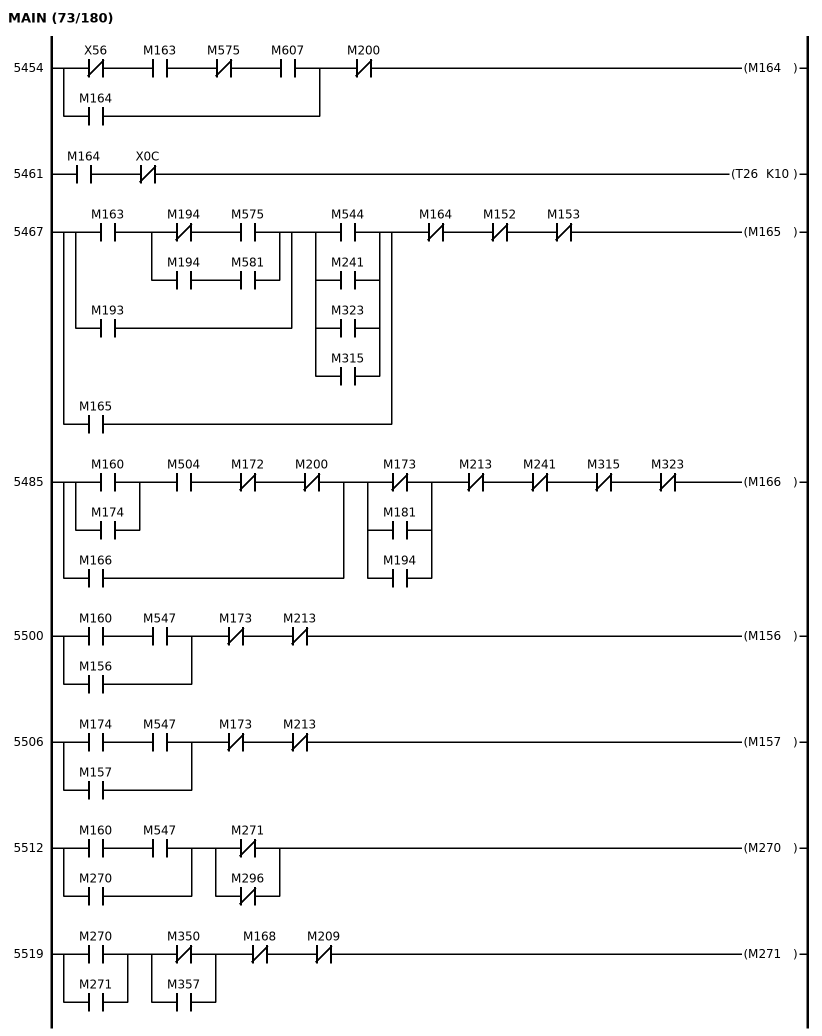
[picture p72: ladder of MAIN, rungs at steps 5454 to 5519]
5454  LDI     X56
      AND     M163
      ANI     M575
      AND     M607
      OR      M164
      ANI     M200
      OUT     M164
5461  LD      M164
      ANI     X0C
      OUT     T26 K10
5467  LD      M163
      LDI     M194
      AND     M575
      LD      M194
      AND     M581
      ORB
      ANB
      OR      M193
      LD      M544
      OR      M241
      OR      M323
      OR      M315
      ANB
      OR      M165
      ANI     M164
      ANI     M152
      ANI     M153
      OUT     M165
5485  LD      M160
      OR      M174
      AND     M504
      ANI     M172
      ANI     M200
      OR      M166
      LDI     M173
      OR      M181
      OR      M194
      ANB
      ANI     M213
      ANI     M241
      ANI     M315
      ANI     M323
      OUT     M166
5500  LD      M160
      AND     M547
      OR      M156
      ANI     M173
      ANI     M213
      OUT     M156
5506  LD      M174
      AND     M547
      OR      M157
      ANI     M173
      ANI     M213
      OUT     M157
5512  LD      M160
      AND     M547
      OR      M270
      LDI     M271
      ORI     M296
      ANB
      OUT     M270
5519  LD      M270
      OR      M271
      LDI     M350
      OR      M357
      ANB
      ANI     M168
      ANI     M209
      OUT     M271
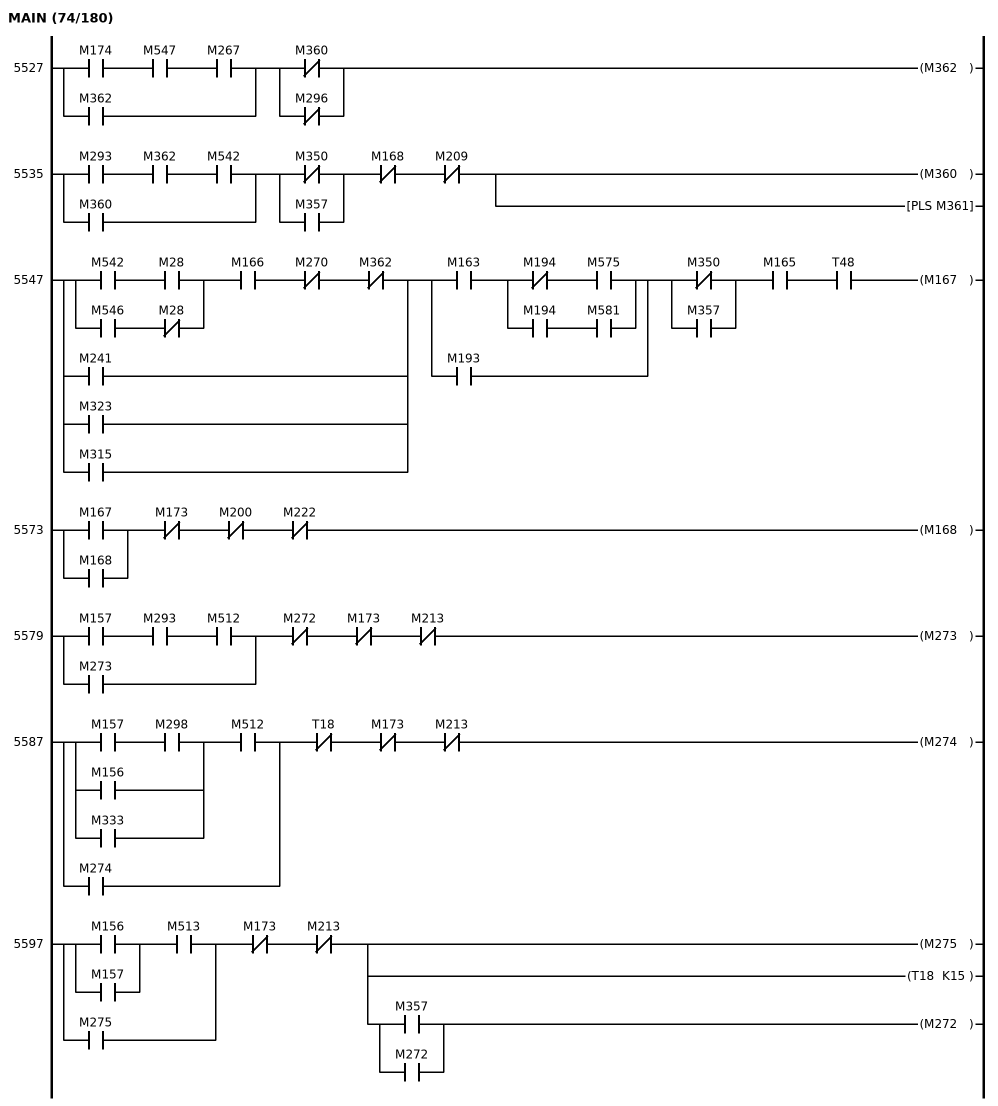
5527  LD      M174
      AND     M547
      AND     M267
      OR      M362
      LDI     M360
      ORI     M296
      ANB
      OUT     M362
5535  LD      M293
      AND     M362
      AND     M542
      OR      M360
      LDI     M350
      OR      M357
      ANB
      ANI     M168
      ANI     M209
      OUT     M360
      PLS     M361
5547  LD      M542
      AND     M28
      LD      M546
      ANI     M28
      ORB
      AND     M166
      ANI     M270
      ANI     M362
      OR      M241
      OR      M323
      OR      M315
      LD      M163
      LDI     M194
      AND     M575
      LD      M194
      AND     M581
      ORB
      ANB
      OR      M193
      ANB
      LDI     M350
      OR      M357
      ANB
      AND     M165
      AND     T48
      OUT     M167
5573  LD      M167
      OR      M168
      ANI     M173
      ANI     M200
      ANI     M222
      OUT     M168
5579  LD      M157
      AND     M293
      AND     M512
      OR      M273
      ANI     M272
      ANI     M173
      ANI     M213
      OUT     M273
5587  LD      M157
      AND     M298
      OR      M156
      OR      M333
      AND     M512
      OR      M274
      ANI     T18
      ANI     M173
      ANI     M213
      OUT     M274
5597  LD      M156
      OR      M157
      AND     M513
      OR      M275
      ANI     M173
      ANI     M213
      OUT     M275
      OUT     T18 K15
      LD      M357
      OR      M272
      ANB
      OUT     M272
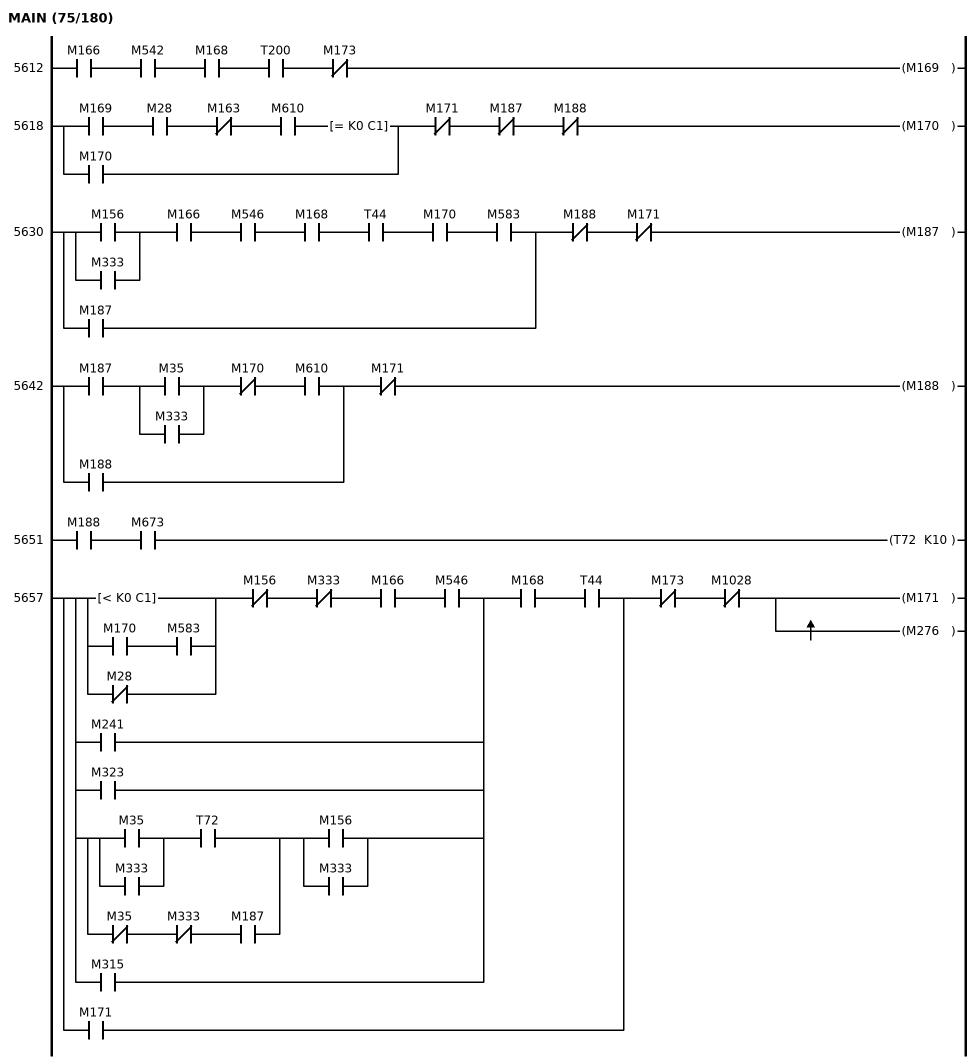
5612  LD      M166
      AND     M542
      AND     M168
      AND     T200
      ANI     M173
      OUT     M169
5618  LD      M169
      AND     M28
      ANI     M163
      AND     M610
      AND=    K0 C1
      OR      M170
      ANI     M171
      ANI     M187
      ANI     M188
      OUT     M170
5630  LD      M156
      OR      M333
      AND     M166
      AND     M546
      AND     M168
      AND     T44
      AND     M170
      AND     M583
      OR      M187
      ANI     M188
      ANI     M171
      OUT     M187
5642  LD      M187
      LD      M35
      OR      M333
      ANB
      ANI     M170
      AND     M610
      OR      M188
      ANI     M171
      OUT     M188
5651  LD      M188
      AND     M673
      OUT     T72 K10
5657  LD<     K0 C1
      LD      M170
      AND     M583
      ORB
      ORI     M28
      ANI     M156
      ANI     M333
      AND     M166
      AND     M546
      OR      M241
      OR      M323
      LD      M35
      OR      M333
      AND     T72
      LDI     M35
      ANI     M333
      AND     M187
      ORB
      LD      M156
      OR      M333
      ANB
      ORB
      OR      M315
      AND     M168
      AND     T44
      OR      M171
      ANI     M173
      ANI     M1028
      OUT     M171
      MEP
      OUT     M276
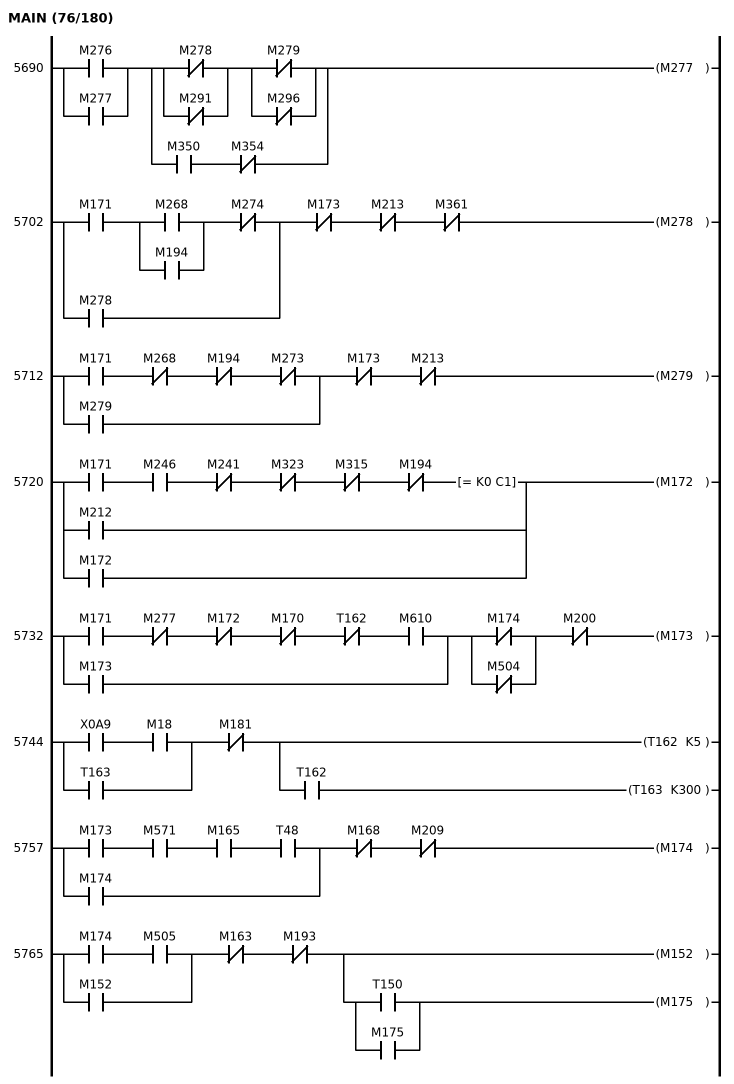
5690  LD      M276
      OR      M277
      LDI     M278
      ORI     M291
      LDI     M279
      ORI     M296
      ANB
      LD      M350
      ANI     M354
      ORB
      ANB
      OUT     M277
5702  LD      M171
      LD      M268
      OR      M194
      ANB
      ANI     M274
      OR      M278
      ANI     M173
      ANI     M213
      ANI     M361
      OUT     M278
5712  LD      M171
      ANI     M268
      ANI     M194
      ANI     M273
      OR      M279
      ANI     M173
      ANI     M213
      OUT     M279
5720  LD      M171
      AND     M246
      ANI     M241
      ANI     M323
      ANI     M315
      ANI     M194
      AND=    K0 C1
      OR      M212
      OR      M172
      OUT     M172
5732  LD      M171
      ANI     M277
      ANI     M172
      ANI     M170
      ANI     T162
      AND     M610
      OR      M173
      LDI     M174
      ORI     M504
      ANB
      ANI     M200
      OUT     M173
5744  LD      X0A9
      AND     M18
      OR      T163
      ANI     M181
      OUT     T162 K5
      AND     T162
      OUT     T163 K300
5757  LD      M173
      AND     M571
      AND     M165
      AND     T48
      OR      M174
      ANI     M168
      ANI     M209
      OUT     M174
5765  LD      M174
      AND     M505
      OR      M152
      ANI     M163
      ANI     M193
      OUT     M152
      LD      T150
      OR      M175
      ANB
      OUT     M175
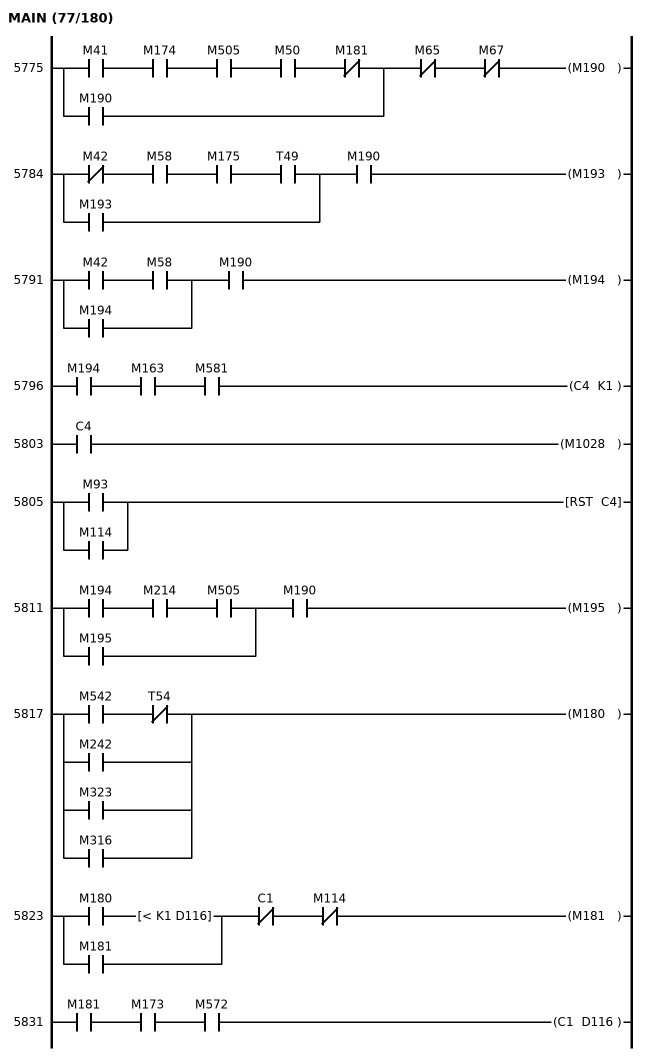
5775  LD      M41
      AND     M174
      AND     M505
      AND     M50
      ANI     M181
      OR      M190
      ANI     M65
      ANI     M67
      OUT     M190
5784  LDI     M42
      AND     M58
      AND     M175
      AND     T49
      OR      M193
      AND     M190
      OUT     M193
5791  LD      M42
      AND     M58
      OR      M194
      AND     M190
      OUT     M194
5796  LD      M194
      AND     M163
      AND     M581
      OUT     C4 K1
5803  LD      C4
      OUT     M1028
5805  LD      M93
      OR      M114
      RST     C4
5811  LD      M194
      AND     M214
      AND     M505
      OR      M195
      AND     M190
      OUT     M195
5817  LD      M542
      ANI     T54
      OR      M242
      OR      M323
      OR      M316
      OUT     M180
5823  LD      M180
      AND<    K1 D116
      OR      M181
      ANI     C1
      ANI     M114
      OUT     M181
5831  LD      M181
      AND     M173
      AND     M572
      OUT     C1 D116
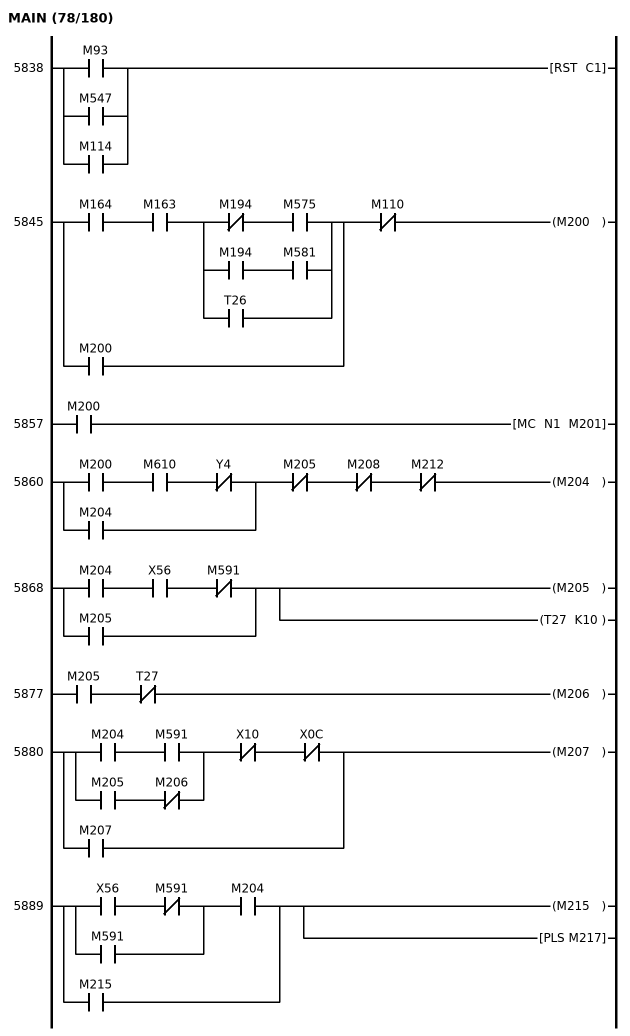
5838  LD      M93
      OR      M547
      OR      M114
      RST     C1
5845  LD      M164
      AND     M163
      LDI     M194
      AND     M575
      LD      M194
      AND     M581
      ORB
      OR      T26
      ANB
      OR      M200
      ANI     M110
      OUT     M200
5857  LD      M200
      MC      N1 M201
5860  LD      M200
      AND     M610
      ANI     Y4
      OR      M204
      ANI     M205
      ANI     M208
      ANI     M212
      OUT     M204
5868  LD      M204
      AND     X56
      ANI     M591
      OR      M205
      OUT     M205
      OUT     T27 K10
5877  LD      M205
      ANI     T27
      OUT     M206
5880  LD      M204
      AND     M591
      LD      M205
      ANI     M206
      ORB
      ANI     X10
      ANI     X0C
      OR      M207
      OUT     M207
5889  LD      X56
      ANI     M591
      OR      M591
      AND     M204
      OR      M215
      OUT     M215
      PLS     M217
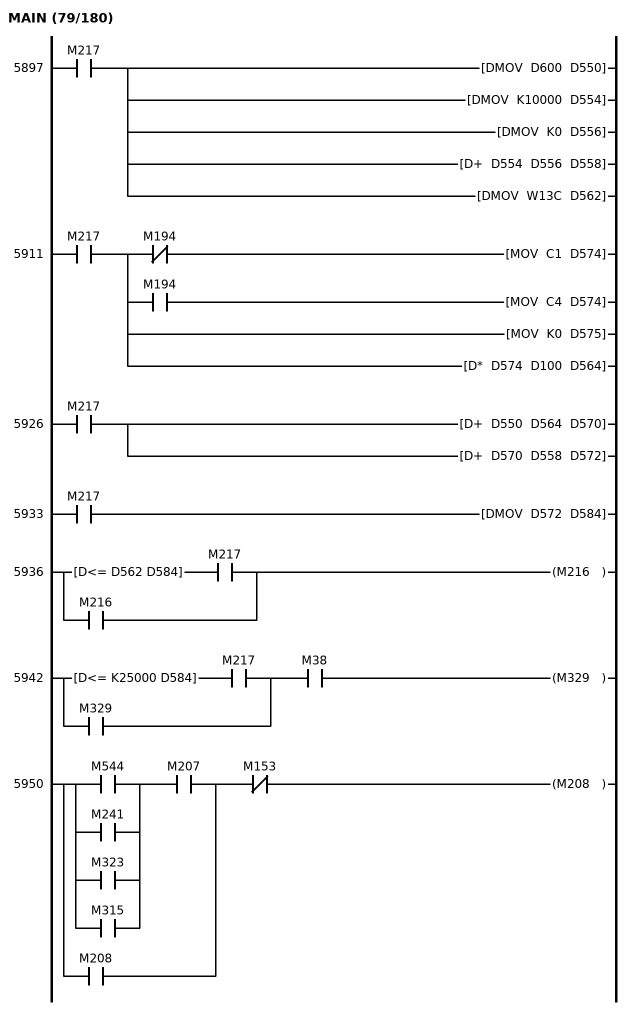
5897  LD      M217
      DMOV    D600 D550
      DMOV    K10000 D554
      DMOV    K0 D556
      D+      D554 D556 D558
      DMOV    W13C D562
5911  LD      M217
      MPS
      ANI     M194
      MOV     C1 D574
      MRD
      AND     M194
      MOV     C4 D574
      MPP
      MOV     K0 D575
      D*      D574 D100 D564
5926  LD      M217
      D+      D550 D564 D570
      D+      D570 D558 D572
5933  LD      M217
      DMOV    D572 D584
5936  LDD<=   D562 D584
      AND     M217
      OR      M216
      OUT     M216
5942  LDD<=   K25000 D584
      AND     M217
      OR      M329
      AND     M38
      OUT     M329
5950  LD      M544
      OR      M241
      OR      M323
      OR      M315
      AND     M207
      OR      M208
      ANI     M153
      OUT     M208
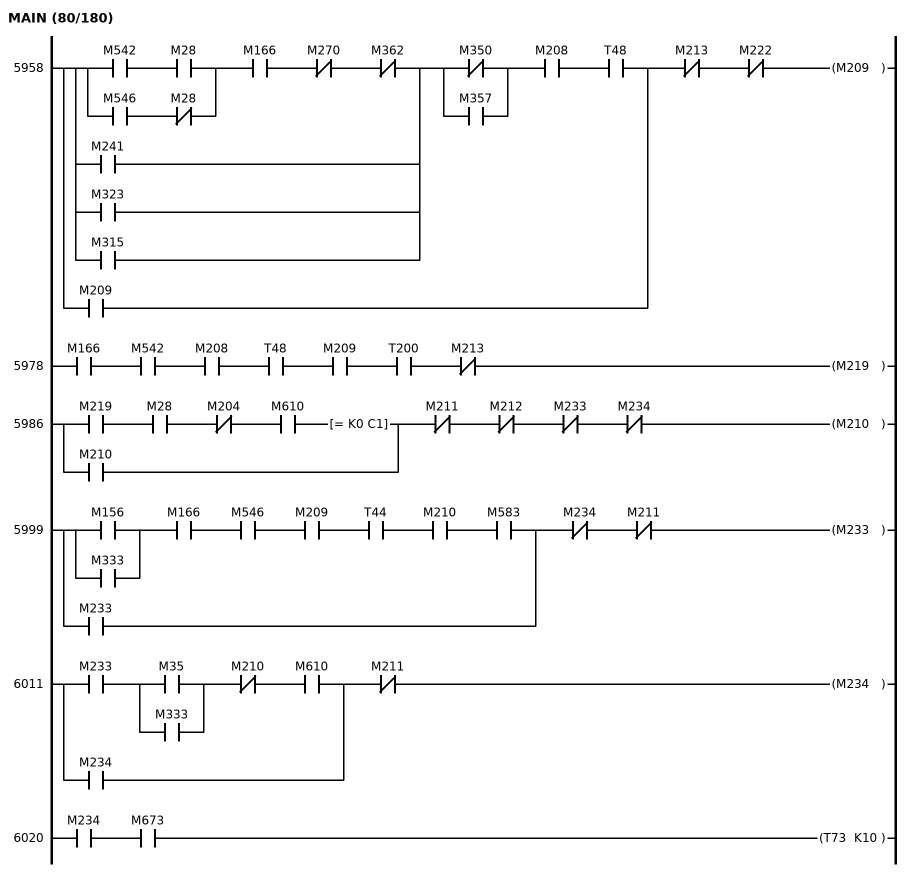
5958  LD      M542
      AND     M28
      LD      M546
      ANI     M28
      ORB
      AND     M166
      ANI     M270
      ANI     M362
      OR      M241
      OR      M323
      OR      M315
      LDI     M350
      OR      M357
      ANB
      AND     M208
      AND     T48
      OR      M209
      ANI     M213
      ANI     M222
      OUT     M209
5978  LD      M166
      AND     M542
      AND     M208
      AND     T48
      AND     M209
      AND     T200
      ANI     M213
      OUT     M219
5986  LD      M219
      AND     M28
      ANI     M204
      AND     M610
      AND=    K0 C1
      OR      M210
      ANI     M211
      ANI     M212
      ANI     M233
      ANI     M234
      OUT     M210
5999  LD      M156
      OR      M333
      AND     M166
      AND     M546
      AND     M209
      AND     T44
      AND     M210
      AND     M583
      OR      M233
      ANI     M234
      ANI     M211
      OUT     M233
6011  LD      M233
      LD      M35
      OR      M333
      ANB
      ANI     M210
      AND     M610
      OR      M234
      ANI     M211
      OUT     M234
6020  LD      M234
      AND     M673
      OUT     T73 K10
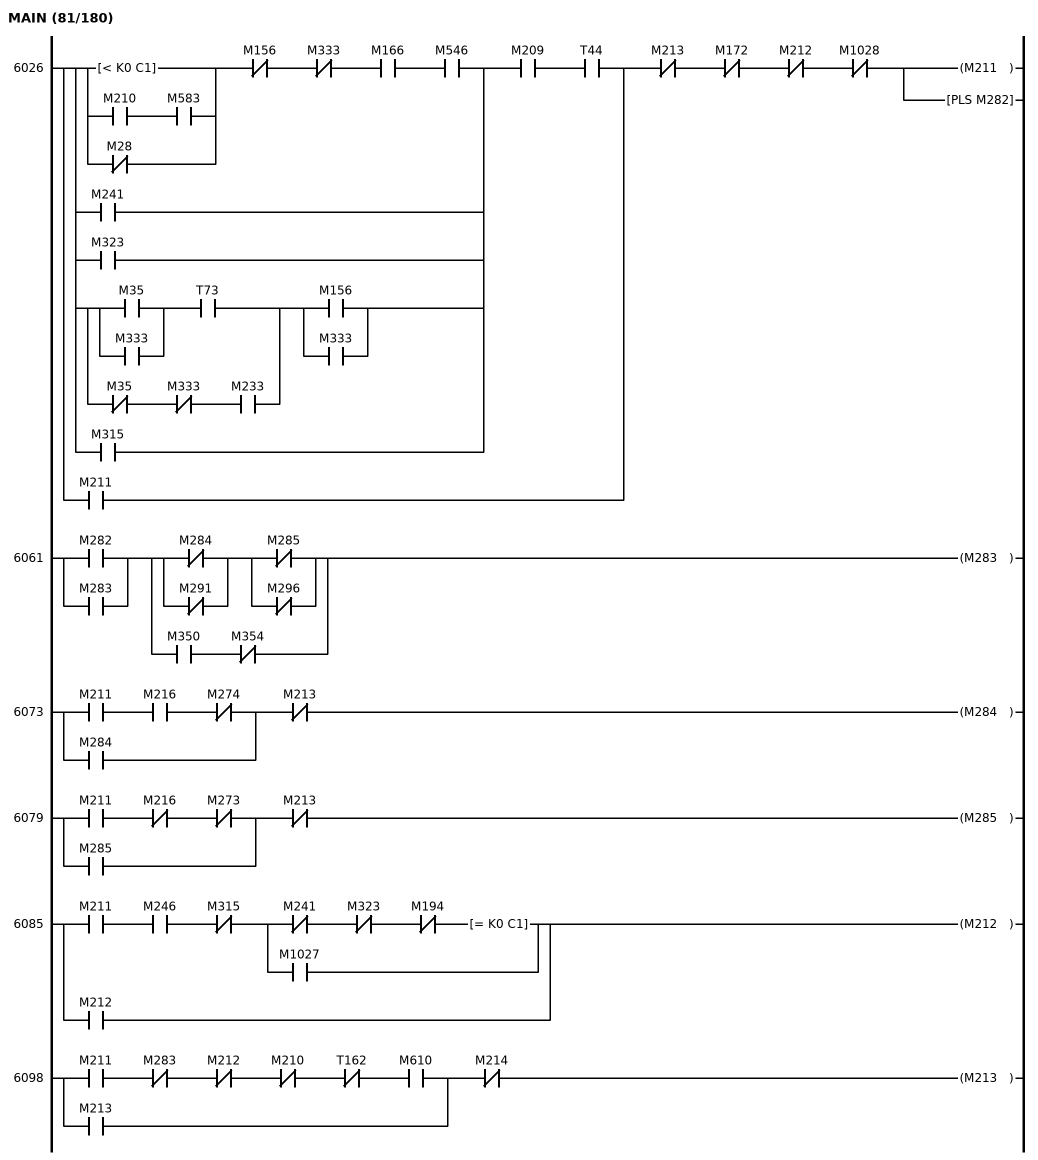
6026  LD<     K0 C1
      LD      M210
      AND     M583
      ORB
      ORI     M28
      ANI     M156
      ANI     M333
      AND     M166
      AND     M546
      OR      M241
      OR      M323
      LD      M35
      OR      M333
      AND     T73
      LDI     M35
      ANI     M333
      AND     M233
      ORB
      LD      M156
      OR      M333
      ANB
      ORB
      OR      M315
      AND     M209
      AND     T44
      OR      M211
      ANI     M213
      ANI     M172
      ANI     M212
      ANI     M1028
      OUT     M211
      PLS     M282
6061  LD      M282
      OR      M283
      LDI     M284
      ORI     M291
      LDI     M285
      ORI     M296
      ANB
      LD      M350
      ANI     M354
      ORB
      ANB
      OUT     M283
6073  LD      M211
      AND     M216
      ANI     M274
      OR      M284
      ANI     M213
      OUT     M284
6079  LD      M211
      ANI     M216
      ANI     M273
      OR      M285
      ANI     M213
      OUT     M285
6085  LD      M211
      AND     M246
      ANI     M315
      LDI     M241
      ANI     M323
      ANI     M194
      AND=    K0 C1
      OR      M1027
      ANB
      OR      M212
      OUT     M212
6098  LD      M211
      ANI     M283
      ANI     M212
      ANI     M210
      ANI     T162
      AND     M610
      OR      M213
      ANI     M214
      OUT     M213
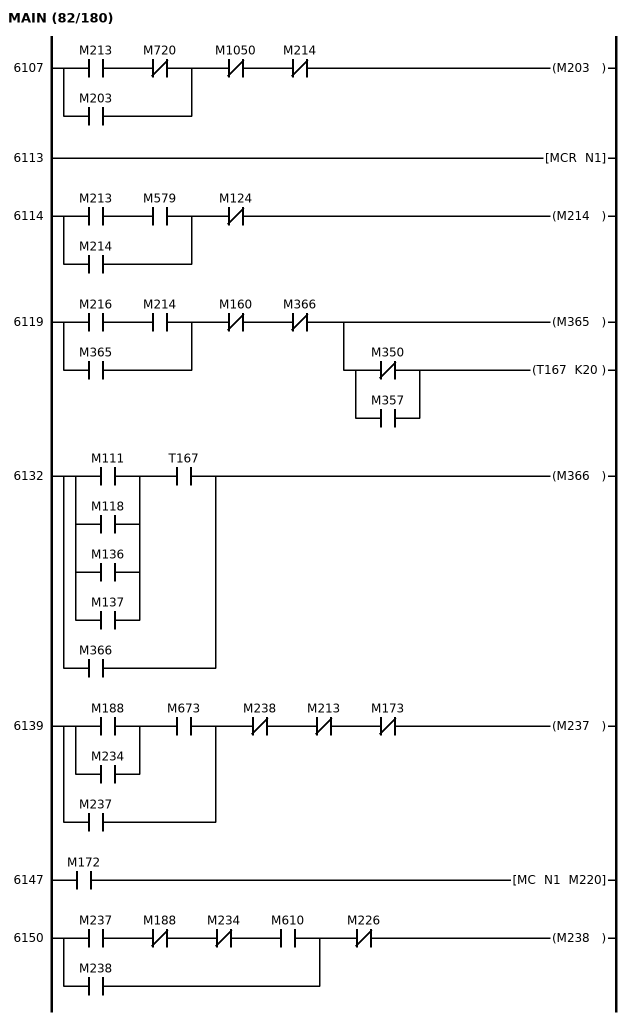
6107  LD      M213
      ANI     M720
      OR      M203
      ANI     M1050
      ANI     M214
      OUT     M203
6113  MCR     N1
6114  LD      M213
      AND     M579
      OR      M214
      ANI     M124
      OUT     M214
6119  LD      M216
      AND     M214
      OR      M365
      ANI     M160
      ANI     M366
      OUT     M365
      LDI     M350
      OR      M357
      ANB
      OUT     T167 K20
6132  LD      M111
      OR      M118
      OR      M136
      OR      M137
      AND     T167
      OR      M366
      OUT     M366
6139  LD      M188
      OR      M234
      AND     M673
      OR      M237
      ANI     M238
      ANI     M213
      ANI     M173
      OUT     M237
6147  LD      M172
      MC      N1 M220
6150  LD      M237
      ANI     M188
      ANI     M234
      AND     M610
      OR      M238
      ANI     M226
      OUT     M238
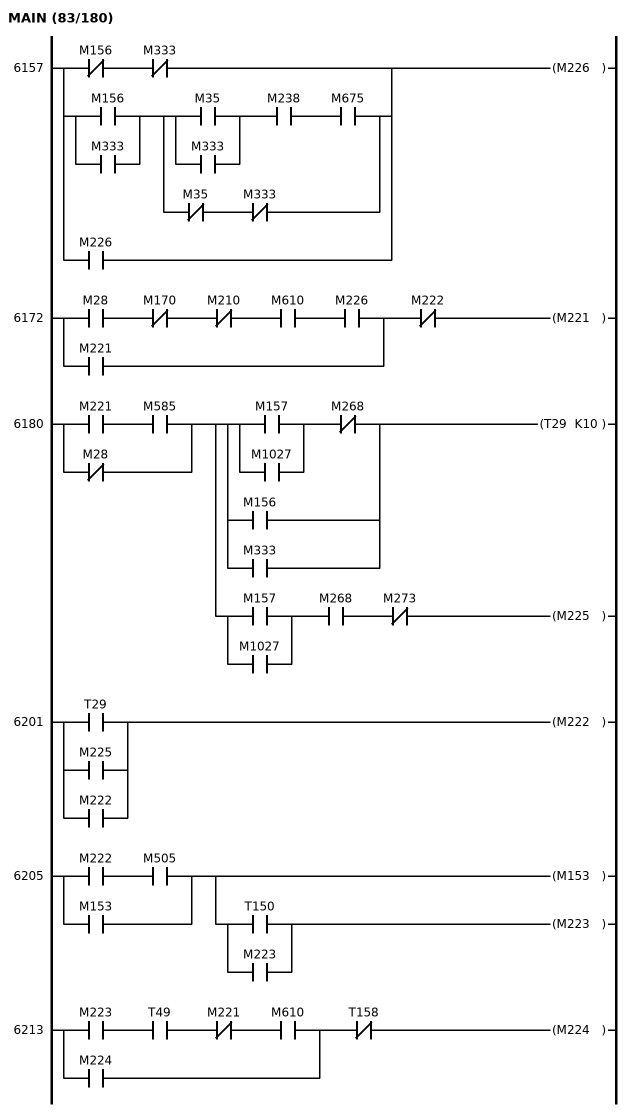
6157  LDI     M156
      ANI     M333
      LD      M156
      OR      M333
      LD      M35
      OR      M333
      AND     M238
      AND     M675
      LDI     M35
      ANI     M333
      ORB
      ANB
      ORB
      OR      M226
      OUT     M226
6172  LD      M28
      ANI     M170
      ANI     M210
      AND     M610
      AND     M226
      OR      M221
      ANI     M222
      OUT     M221
6180  LD      M221
      AND     M585
      ORI     M28
      MPS
      LD      M157
      OR      M1027
      ANI     M268
      OR      M156
      OR      M333
      ANB
      OUT     T29 K10
      MPP
      LD      M157
      OR      M1027
      ANB
      AND     M268
      ANI     M273
      OUT     M225
6201  LD      T29
      OR      M225
      OR      M222
      OUT     M222
6205  LD      M222
      AND     M505
      OR      M153
      OUT     M153
      LD      T150
      OR      M223
      ANB
      OUT     M223
6213  LD      M223
      AND     T49
      ANI     M221
      AND     M610
      OR      M224
      ANI     T158
      OUT     M224
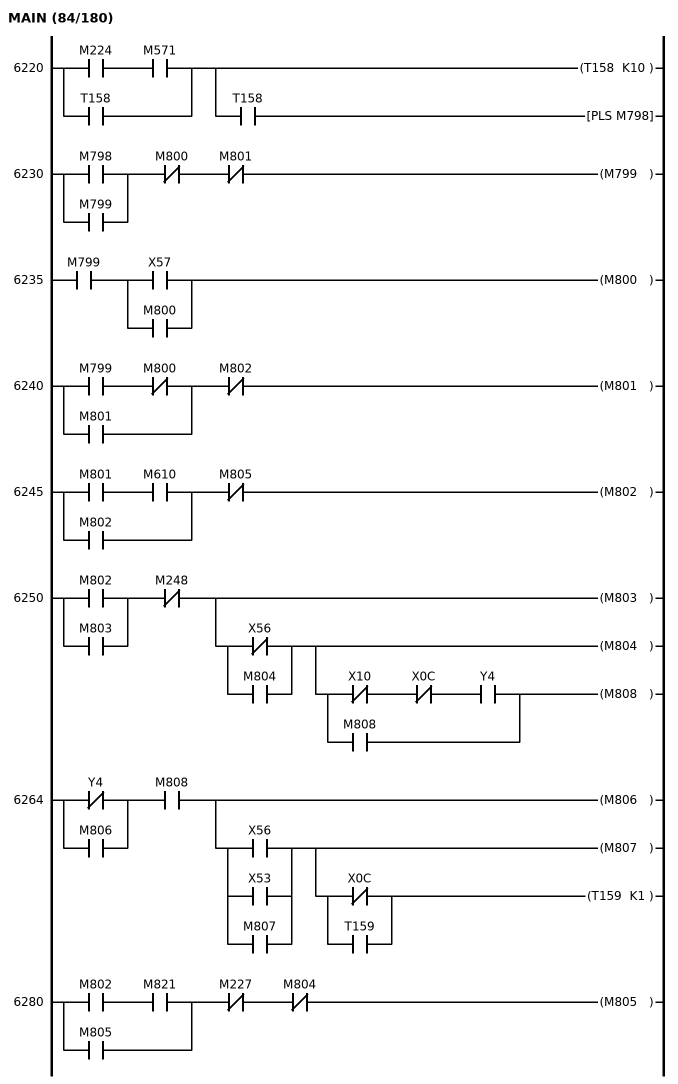
6220  LD      M224
      AND     M571
      OR      T158
      OUT     T158 K10
      AND     T158
      PLS     M798
6230  LD      M798
      OR      M799
      ANI     M800
      ANI     M801
      OUT     M799
6235  LD      M799
      LD      X57
      OR      M800
      ANB
      OUT     M800
6240  LD      M799
      ANI     M800
      OR      M801
      ANI     M802
      OUT     M801
6245  LD      M801
      AND     M610
      OR      M802
      ANI     M805
      OUT     M802
6250  LD      M802
      OR      M803
      ANI     M248
      OUT     M803
      LDI     X56
      OR      M804
      ANB
      OUT     M804
      LDI     X10
      ANI     X0C
      AND     Y4
      OR      M808
      ANB
      OUT     M808
6264  LDI     Y4
      OR      M806
      AND     M808
      OUT     M806
      LD      X56
      OR      X53
      OR      M807
      ANB
      OUT     M807
      LDI     X0C
      OR      T159
      ANB
      OUT     T159 K1
6280  LD      M802
      AND     M821
      OR      M805
      ANI     M227
      ANI     M804
      OUT     M805
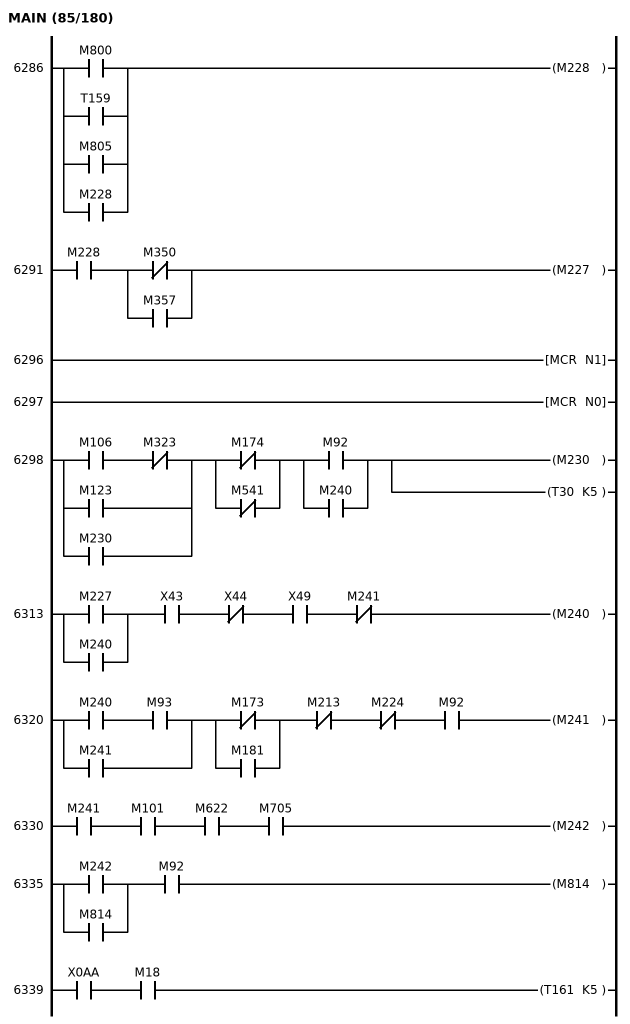
6286  LD      M800
      OR      T159
      OR      M805
      OR      M228
      OUT     M228
6291  LD      M228
      LDI     M350
      OR      M357
      ANB
      OUT     M227
6296  MCR     N1
6297  MCR     N0
6298  LD      M106
      ANI     M323
      OR      M123
      OR      M230
      LDI     M174
      ORI     M541
      ANB
      LD      M92
      OR      M240
      ANB
      OUT     M230
      OUT     T30 K5
6313  LD      M227
      OR      M240
      AND     X43
      ANI     X44
      AND     X49
      ANI     M241
      OUT     M240
6320  LD      M240
      AND     M93
      OR      M241
      LDI     M173
      OR      M181
      ANB
      ANI     M213
      ANI     M224
      AND     M92
      OUT     M241
6330  LD      M241
      AND     M101
      AND     M622
      AND     M705
      OUT     M242
6335  LD      M242
      OR      M814
      AND     M92
      OUT     M814
6339  LD      X0AA
      AND     M18
      OUT     T161 K5
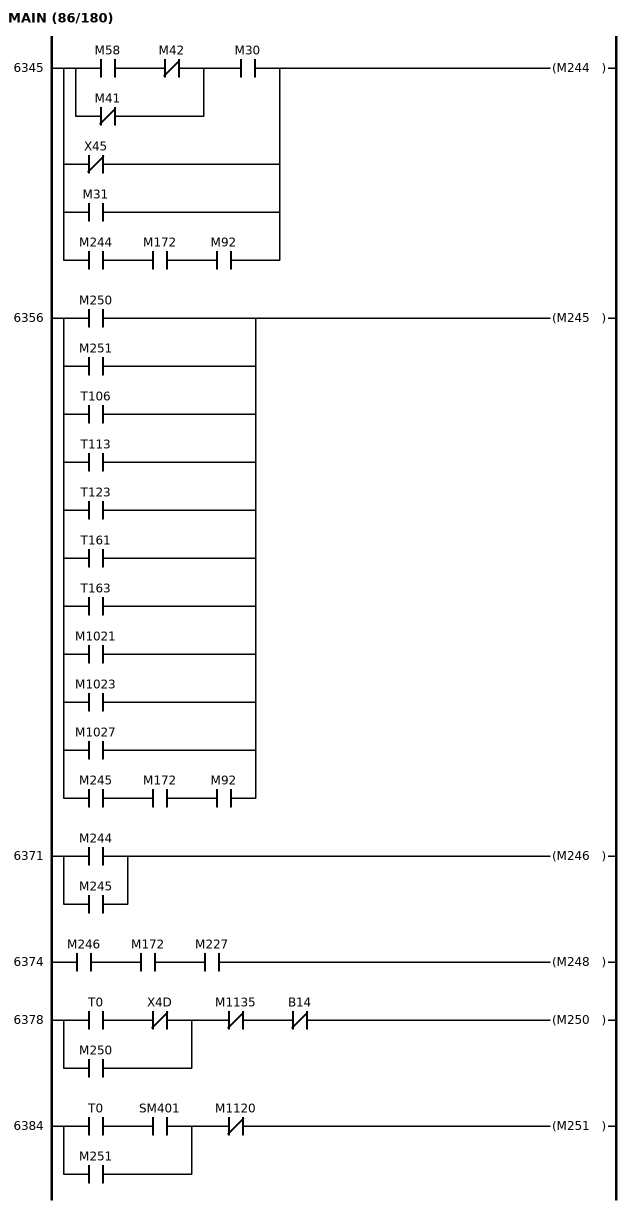
6345  LD      M58
      ANI     M42
      ORI     M41
      AND     M30
      ORI     X45
      OR      M31
      LD      M244
      AND     M172
      AND     M92
      ORB
      OUT     M244
6356  LD      M250
      OR      M251
      OR      T106
      OR      T113
      OR      T123
      OR      T161
      OR      T163
      OR      M1021
      OR      M1023
      OR      M1027
      LD      M245
      AND     M172
      AND     M92
      ORB
      OUT     M245
6371  LD      M244
      OR      M245
      OUT     M246
6374  LD      M246
      AND     M172
      AND     M227
      OUT     M248
6378  LD      T0
      ANI     X4D
      OR      M250
      ANI     M1135
      ANI     B14
      OUT     M250
6384  LD      T0
      AND     SM401
      OR      M251
      ANI     M1120
      OUT     M251
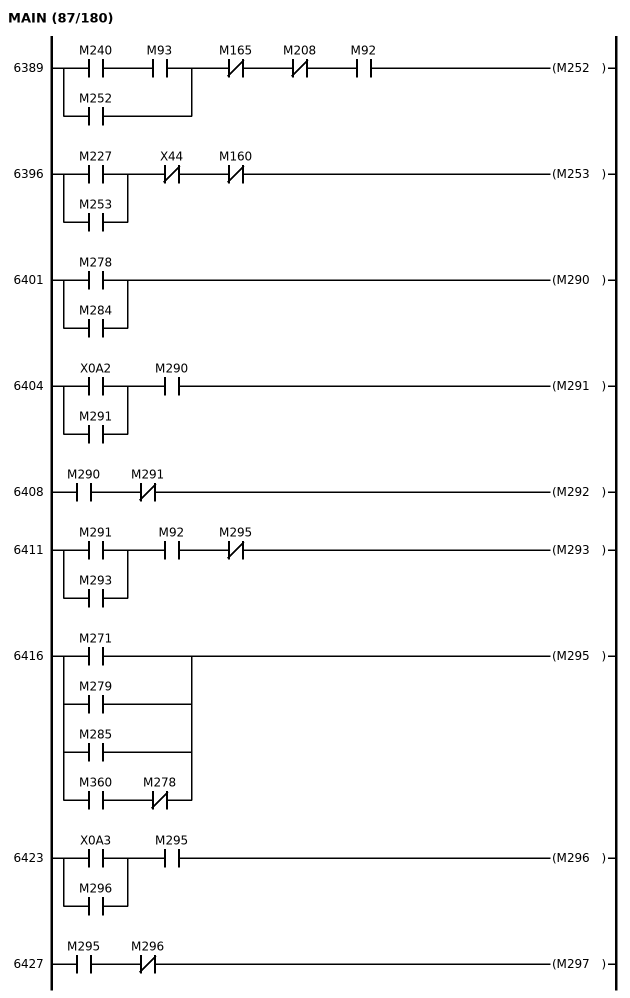
6389  LD      M240
      AND     M93
      OR      M252
      ANI     M165
      ANI     M208
      AND     M92
      OUT     M252
6396  LD      M227
      OR      M253
      ANI     X44
      ANI     M160
      OUT     M253
6401  LD      M278
      OR      M284
      OUT     M290
6404  LD      X0A2
      OR      M291
      AND     M290
      OUT     M291
6408  LD      M290
      ANI     M291
      OUT     M292
6411  LD      M291
      OR      M293
      AND     M92
      ANI     M295
      OUT     M293
6416  LD      M271
      OR      M279
      OR      M285
      LD      M360
      ANI     M278
      ORB
      OUT     M295
6423  LD      X0A3
      OR      M296
      AND     M295
      OUT     M296
6427  LD      M295
      ANI     M296
      OUT     M297
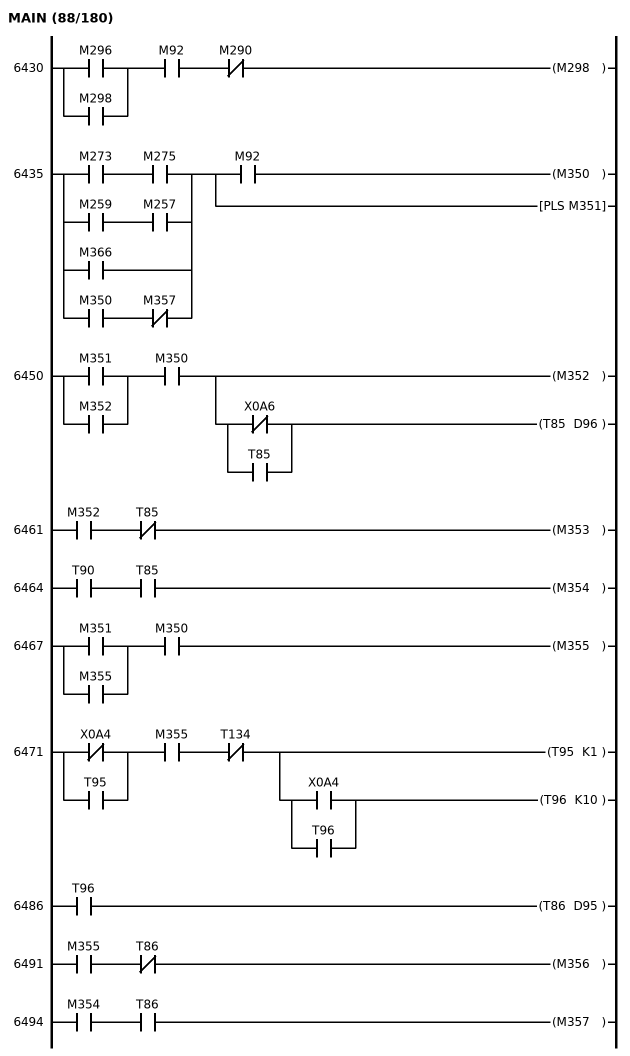
6430  LD      M296
      OR      M298
      AND     M92
      ANI     M290
      OUT     M298
6435  LD      M273
      AND     M275
      LD      M259
      AND     M257
      ORB
      OR      M366
      LD      M350
      ANI     M357
      ORB
      MPS
      AND     M92
      OUT     M350
      MPP
      PLS     M351
6450  LD      M351
      OR      M352
      AND     M350
      OUT     M352
      LDI     X0A6
      OR      T85
      ANB
      OUT     T85 D96
6461  LD      M352
      ANI     T85
      OUT     M353
6464  LD      T90
      AND     T85
      OUT     M354
6467  LD      M351
      OR      M355
      AND     M350
      OUT     M355
6471  LDI     X0A4
      OR      T95
      AND     M355
      ANI     T134
      OUT     T95 K1
      LD      X0A4
      OR      T96
      ANB
      OUT     T96 K10
6486  LD      T96
      OUT     T86 D95
6491  LD      M355
      ANI     T86
      OUT     M356
6494  LD      M354
      AND     T86
      OUT     M357
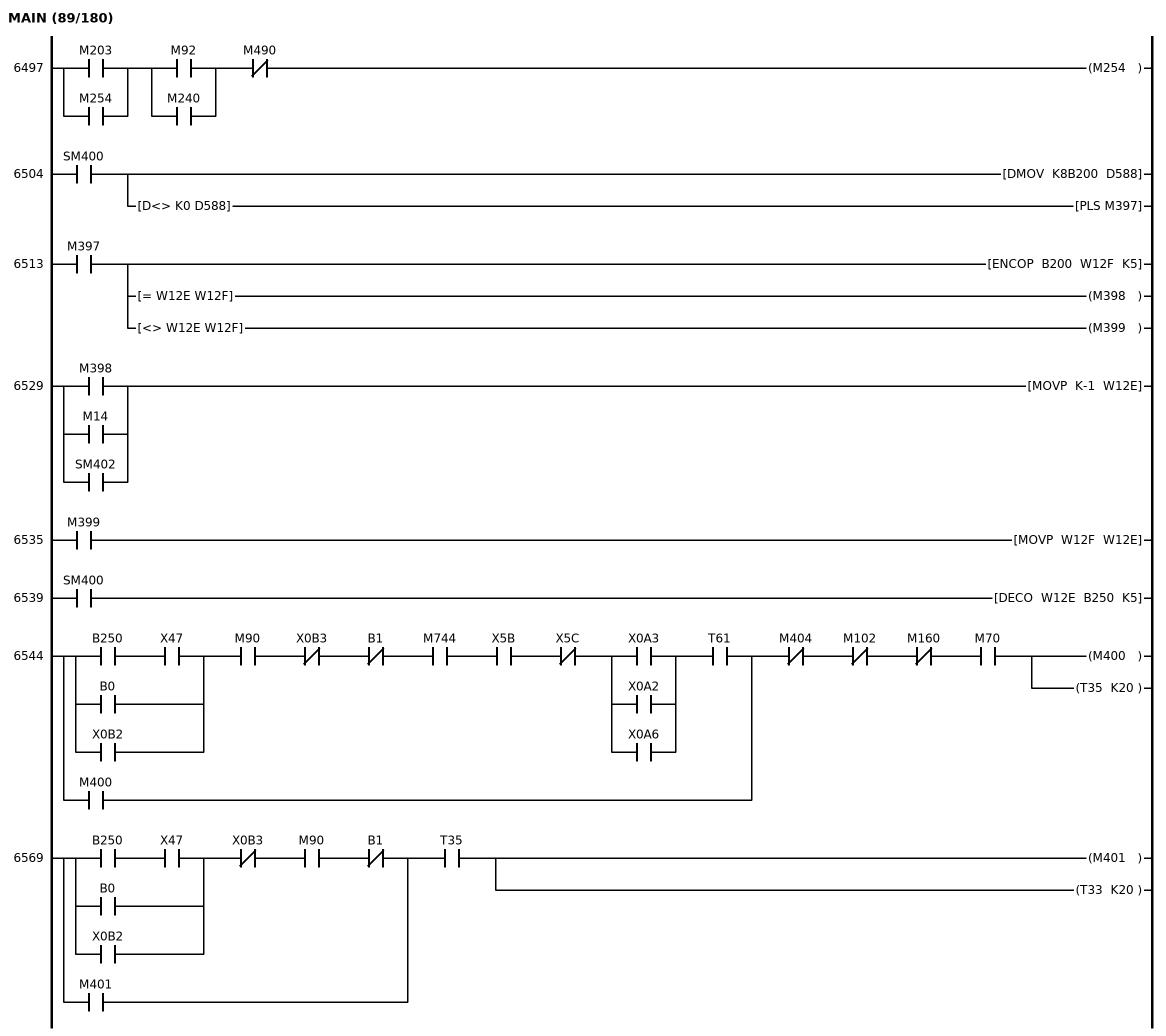
6497  LD      M203
      OR      M254
      LD      M92
      OR      M240
      ANB
      ANI     M490
      OUT     M254
6504  LD      SM400
      DMOV    K8B200 D588
      ANDD<>  K0 D588
      PLS     M397
6513  LD      M397
      ENCOP   B200 W12F K5
      MPS
      AND=    W12E W12F
      OUT     M398
      MPP
      AND<>   W12E W12F
      OUT     M399
6529  LD      M398
      OR      M14
      OR      SM402
      MOVP    K-1 W12E
6535  LD      M399
      MOVP    W12F W12E
6539  LD      SM400
      DECO    W12E B250 K5
6544  LD      B250
      AND     X47
      OR      B0
      OR      X0B2
      AND     M90
      ANI     X0B3
      ANI     B1
      AND     M744
      AND     X5B
      ANI     X5C
      LD      X0A3
      OR      X0A2
      OR      X0A6
      ANB
      AND     T61
      OR      M400
      ANI     M404
      ANI     M102
      ANI     M160
      AND     M70
      OUT     M400
      OUT     T35 K20
6569  LD      B250
      AND     X47
      OR      B0
      OR      X0B2
      ANI     X0B3
      AND     M90
      ANI     B1
      OR      M401
      AND     T35
      OUT     M401
      OUT     T33 K20
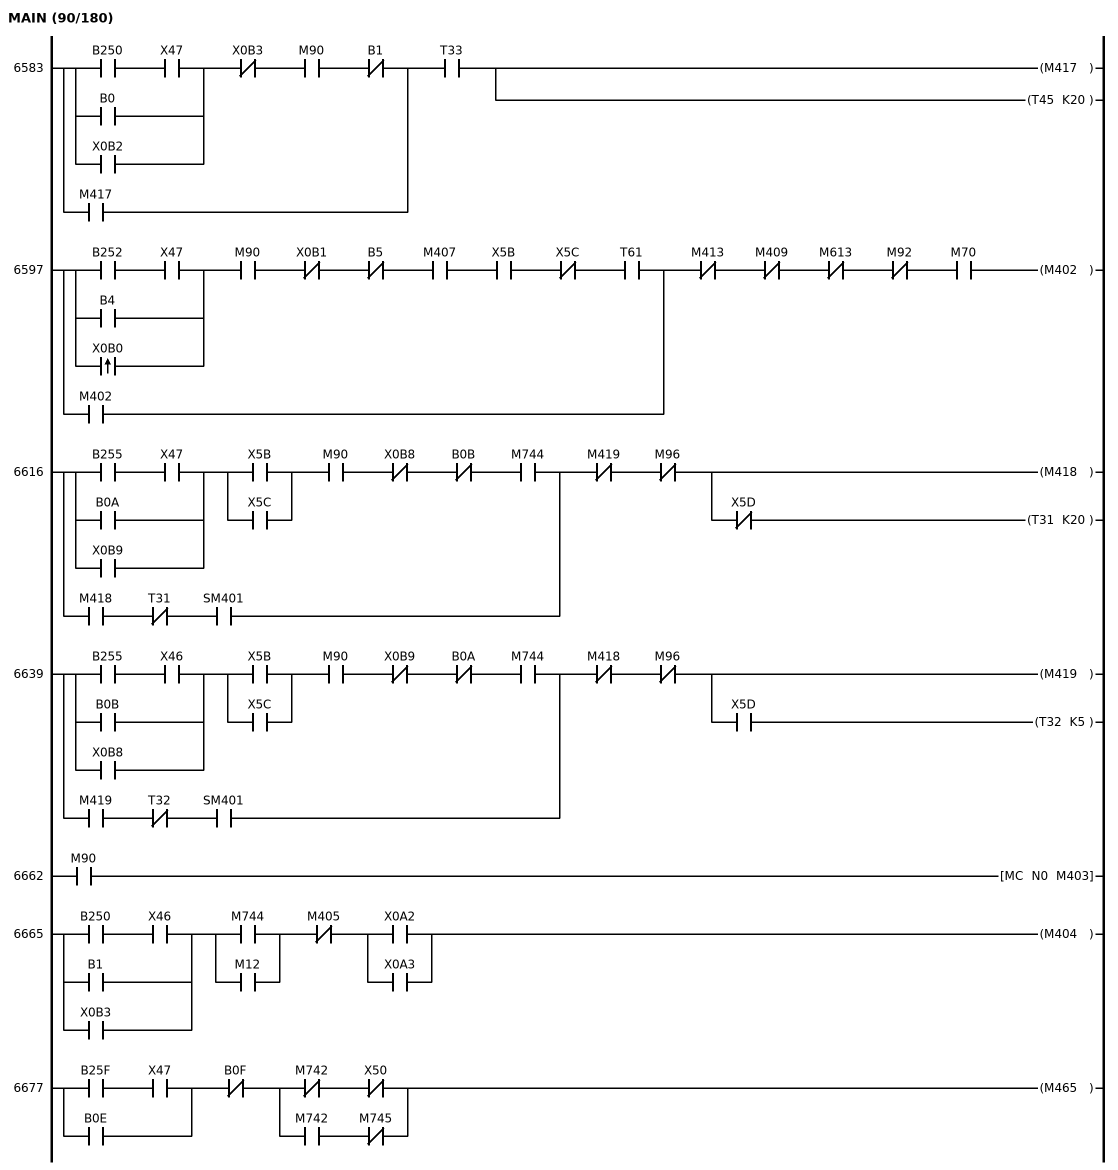
6583  LD      B250
      AND     X47
      OR      B0
      OR      X0B2
      ANI     X0B3
      AND     M90
      ANI     B1
      OR      M417
      AND     T33
      OUT     M417
      OUT     T45 K20
6597  LD      B252
      AND     X47
      OR      B4
      ORP     X0B0
      AND     M90
      ANI     X0B1
      ANI     B5
      AND     M407
      AND     X5B
      ANI     X5C
      AND     T61
      OR      M402
      ANI     M413
      ANI     M409
      ANI     M613
      ANI     M92
      AND     M70
      OUT     M402
6616  LD      B255
      AND     X47
      OR      B0A
      OR      X0B9
      LD      X5B
      OR      X5C
      ANB
      AND     M90
      ANI     X0B8
      ANI     B0B
      AND     M744
      LD      M418
      ANI     T31
      AND     SM401
      ORB
      ANI     M419
      ANI     M96
      OUT     M418
      ANI     X5D
      OUT     T31 K20
6639  LD      B255
      AND     X46
      OR      B0B
      OR      X0B8
      LD      X5B
      OR      X5C
      ANB
      AND     M90
      ANI     X0B9
      ANI     B0A
      AND     M744
      LD      M419
      ANI     T32
      AND     SM401
      ORB
      ANI     M418
      ANI     M96
      OUT     M419
      AND     X5D
      OUT     T32 K5
6662  LD      M90
      MC      N0 M403
6665  LD      B250
      AND     X46
      OR      B1
      OR      X0B3
      LD      M744
      OR      M12
      ANB
      ANI     M405
      LD      X0A2
      OR      X0A3
      ANB
      OUT     M404
6677  LD      B25F
      AND     X47
      OR      B0E
      ANI     B0F
      LDI     M742
      ANI     X50
      LD      M742
      ANI     M745
      ORB
      ANB
      OUT     M465
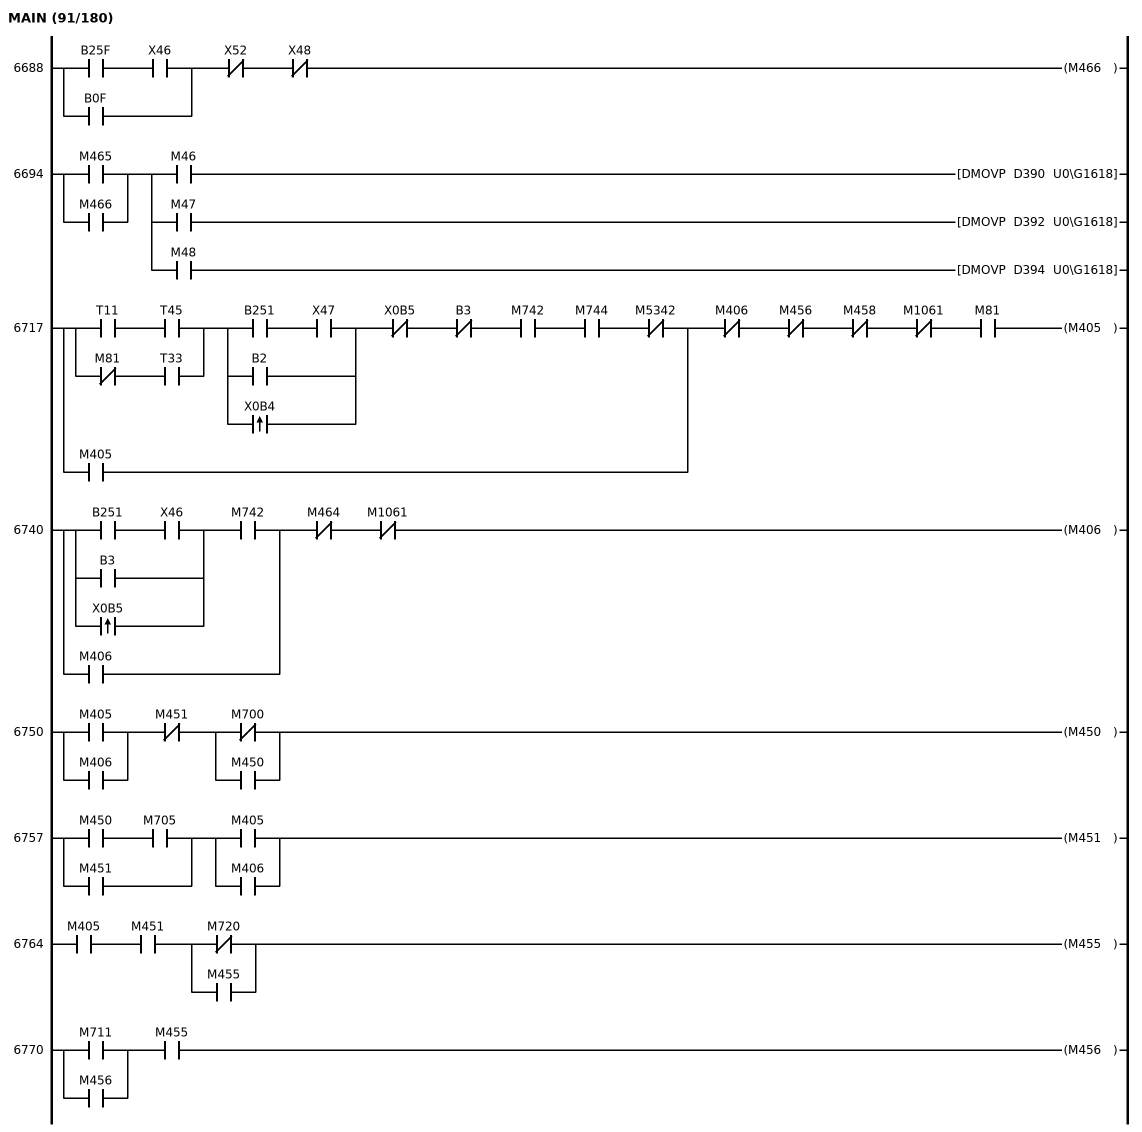
6688  LD      B25F
      AND     X46
      OR      B0F
      ANI     X52
      ANI     X48
      OUT     M466
6694  LD      M465
      OR      M466
      MPS
      AND     M46
      DMOVP   D390 U0\G1618
      MRD
      AND     M47
      DMOVP   D392 U0\G1618
      MPP
      AND     M48
      DMOVP   D394 U0\G1618
6717  LD      T11
      AND     T45
      LDI     M81
      AND     T33
      ORB
      LD      B251
      AND     X47
      OR      B2
      ORP     X0B4
      ANB
      ANI     X0B5
      ANI     B3
      AND     M742
      AND     M744
      ANI     M5342
      OR      M405
      ANI     M406
      ANI     M456
      ANI     M458
      ANI     M1061
      AND     M81
      OUT     M405
6740  LD      B251
      AND     X46
      OR      B3
      ORP     X0B5
      AND     M742
      OR      M406
      ANI     M464
      ANI     M1061
      OUT     M406
6750  LD      M405
      OR      M406
      ANI     M451
      LDI     M700
      OR      M450
      ANB
      OUT     M450
6757  LD      M450
      AND     M705
      OR      M451
      LD      M405
      OR      M406
      ANB
      OUT     M451
6764  LD      M405
      AND     M451
      LDI     M720
      OR      M455
      ANB
      OUT     M455
6770  LD      M711
      OR      M456
      AND     M455
      OUT     M456
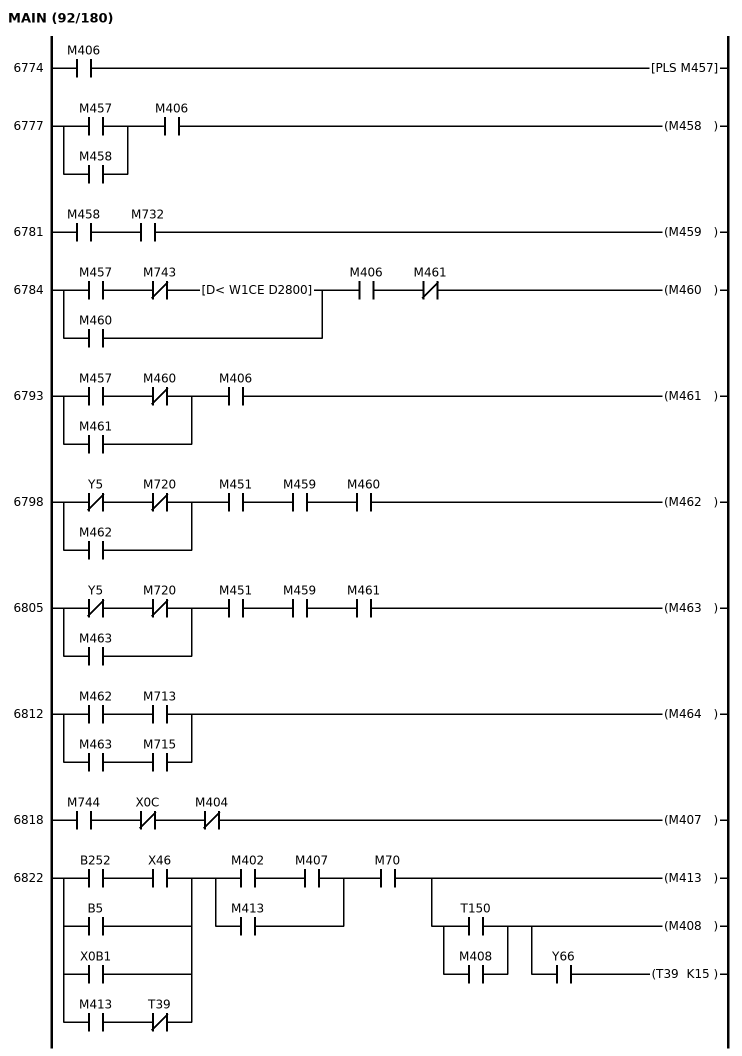
6774  LD      M406
      PLS     M457
6777  LD      M457
      OR      M458
      AND     M406
      OUT     M458
6781  LD      M458
      AND     M732
      OUT     M459
6784  LD      M457
      ANI     M743
      ANDD<   W1CE D2800
      OR      M460
      AND     M406
      ANI     M461
      OUT     M460
6793  LD      M457
      ANI     M460
      OR      M461
      AND     M406
      OUT     M461
6798  LDI     Y5
      ANI     M720
      OR      M462
      AND     M451
      AND     M459
      AND     M460
      OUT     M462
6805  LDI     Y5
      ANI     M720
      OR      M463
      AND     M451
      AND     M459
      AND     M461
      OUT     M463
6812  LD      M462
      AND     M713
      LD      M463
      AND     M715
      ORB
      OUT     M464
6818  LD      M744
      ANI     X0C
      ANI     M404
      OUT     M407
6822  LD      B252
      AND     X46
      OR      B5
      OR      X0B1
      LD      M413
      ANI     T39
      ORB
      LD      M402
      AND     M407
      OR      M413
      ANB
      AND     M70
      OUT     M413
      LD      T150
      OR      M408
      ANB
      OUT     M408
      AND     Y66
      OUT     T39 K15
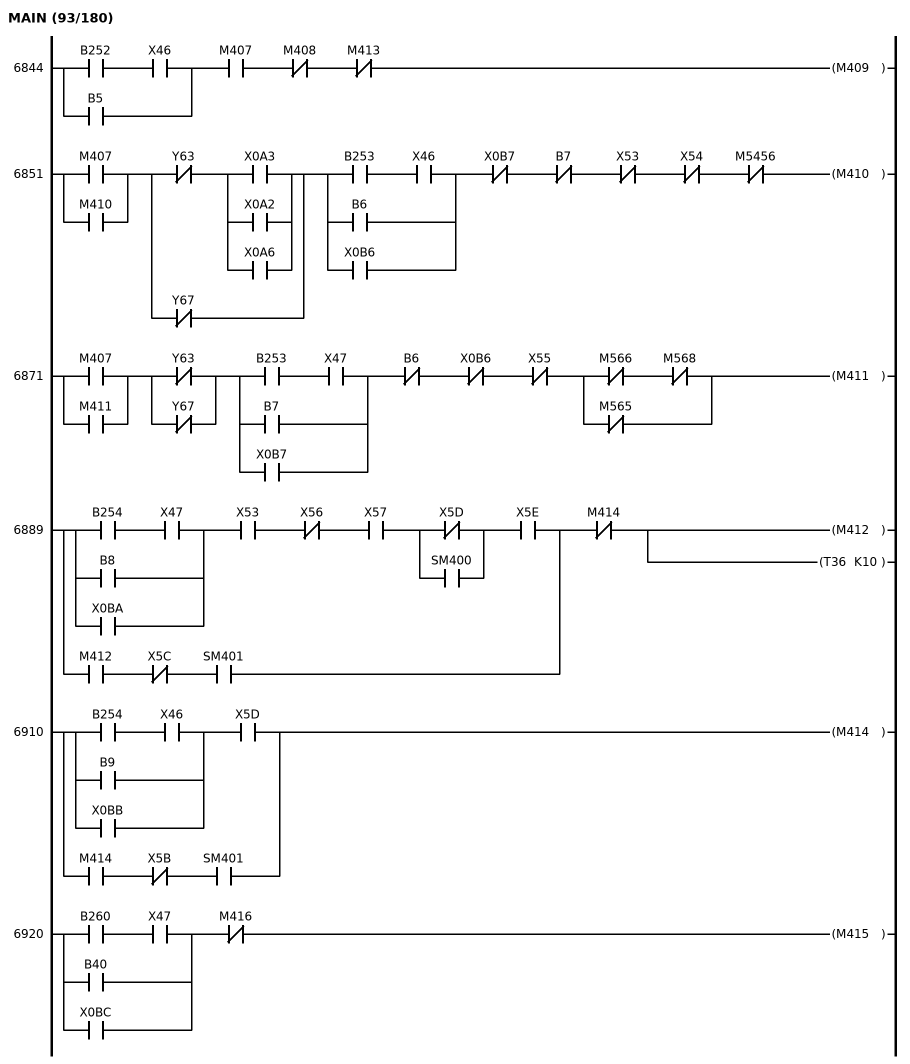
6844  LD      B252
      AND     X46
      OR      B5
      AND     M407
      ANI     M408
      ANI     M413
      OUT     M409
6851  LD      M407
      OR      M410
      LDI     Y63
      LD      X0A3
      OR      X0A2
      OR      X0A6
      ANB
      ORI     Y67
      ANB
      LD      B253
      AND     X46
      OR      B6
      OR      X0B6
      ANB
      ANI     X0B7
      ANI     B7
      ANI     X53
      ANI     X54
      ANI     M5456
      OUT     M410
6871  LD      M407
      OR      M411
      LDI     Y63
      ORI     Y67
      ANB
      LD      B253
      AND     X47
      OR      B7
      OR      X0B7
      ANB
      ANI     B6
      ANI     X0B6
      ANI     X55
      LDI     M566
      ANI     M568
      ORI     M565
      ANB
      OUT     M411
6889  LD      B254
      AND     X47
      OR      B8
      OR      X0BA
      AND     X53
      ANI     X56
      AND     X57
      LDI     X5D
      OR      SM400
      ANB
      AND     X5E
      LD      M412
      ANI     X5C
      AND     SM401
      ORB
      ANI     M414
      OUT     M412
      OUT     T36 K10
6910  LD      B254
      AND     X46
      OR      B9
      OR      X0BB
      AND     X5D
      LD      M414
      ANI     X5B
      AND     SM401
      ORB
      OUT     M414
6920  LD      B260
      AND     X47
      OR      B40
      OR      X0BC
      ANI     M416
      OUT     M415
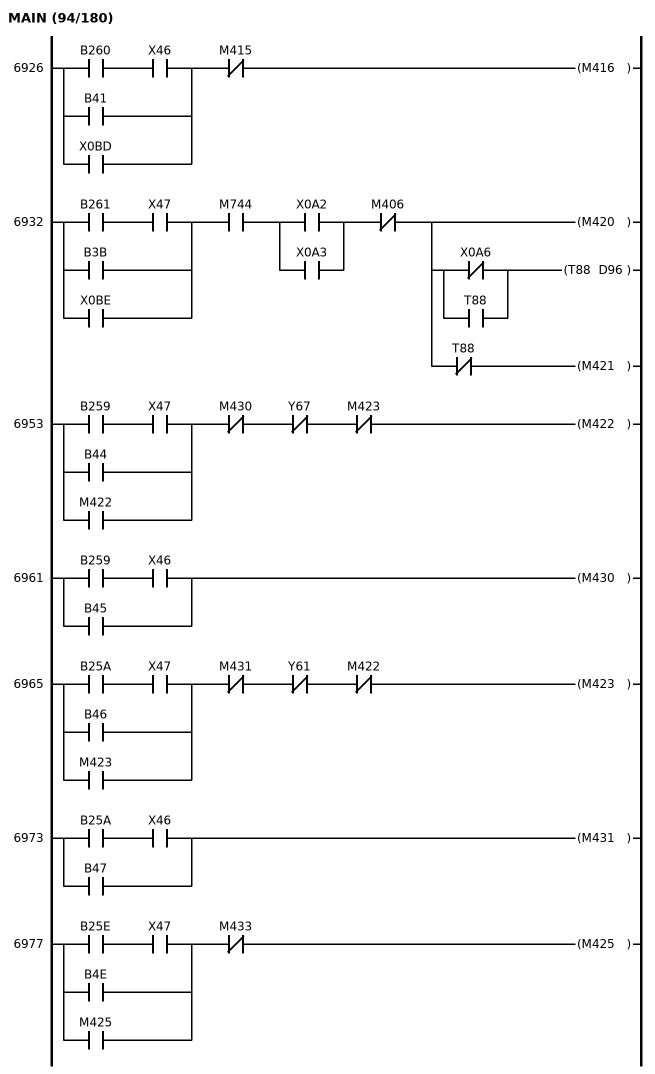
6926  LD      B260
      AND     X46
      OR      B41
      OR      X0BD
      ANI     M415
      OUT     M416
6932  LD      B261
      AND     X47
      OR      B3B
      OR      X0BE
      AND     M744
      LD      X0A2
      OR      X0A3
      ANB
      ANI     M406
      OUT     M420
      MPS
      LDI     X0A6
      OR      T88
      ANB
      OUT     T88 D96
      MPP
      ANI     T88
      OUT     M421
6953  LD      B259
      AND     X47
      OR      B44
      OR      M422
      ANI     M430
      ANI     Y67
      ANI     M423
      OUT     M422
6961  LD      B259
      AND     X46
      OR      B45
      OUT     M430
6965  LD      B25A
      AND     X47
      OR      B46
      OR      M423
      ANI     M431
      ANI     Y61
      ANI     M422
      OUT     M423
6973  LD      B25A
      AND     X46
      OR      B47
      OUT     M431
6977  LD      B25E
      AND     X47
      OR      B4E
      OR      M425
      ANI     M433
      OUT     M425
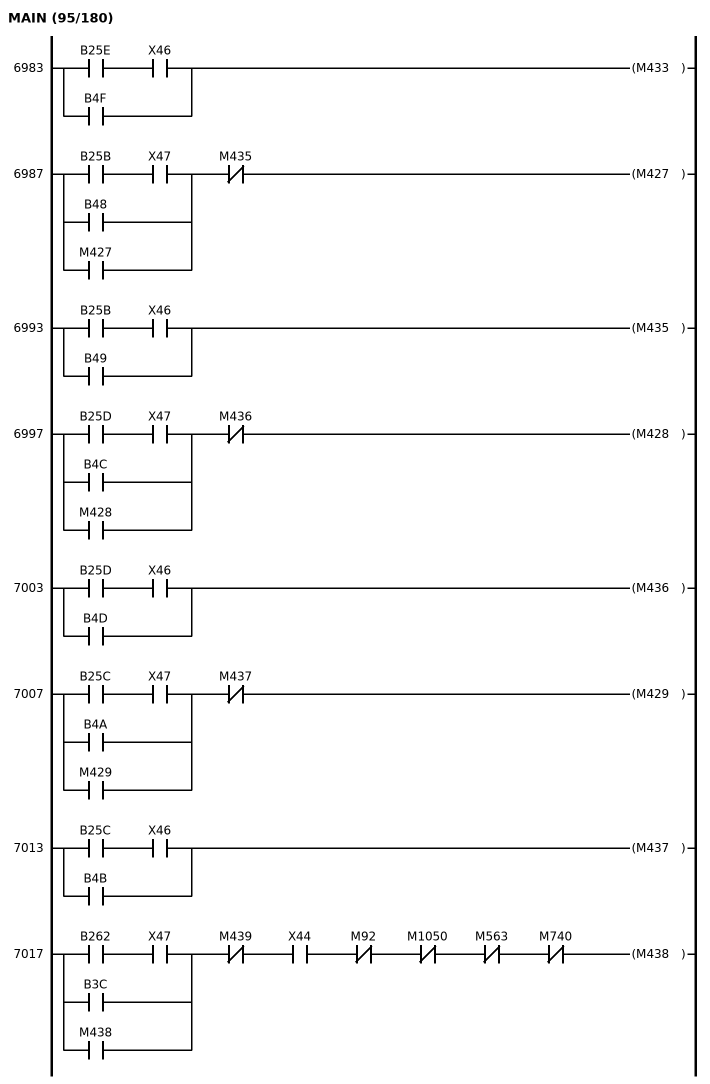
6983  LD      B25E
      AND     X46
      OR      B4F
      OUT     M433
6987  LD      B25B
      AND     X47
      OR      B48
      OR      M427
      ANI     M435
      OUT     M427
6993  LD      B25B
      AND     X46
      OR      B49
      OUT     M435
6997  LD      B25D
      AND     X47
      OR      B4C
      OR      M428
      ANI     M436
      OUT     M428
7003  LD      B25D
      AND     X46
      OR      B4D
      OUT     M436
7007  LD      B25C
      AND     X47
      OR      B4A
      OR      M429
      ANI     M437
      OUT     M429
7013  LD      B25C
      AND     X46
      OR      B4B
      OUT     M437
7017  LD      B262
      AND     X47
      OR      B3C
      OR      M438
      ANI     M439
      AND     X44
      ANI     M92
      ANI     M1050
      ANI     M563
      ANI     M740
      OUT     M438
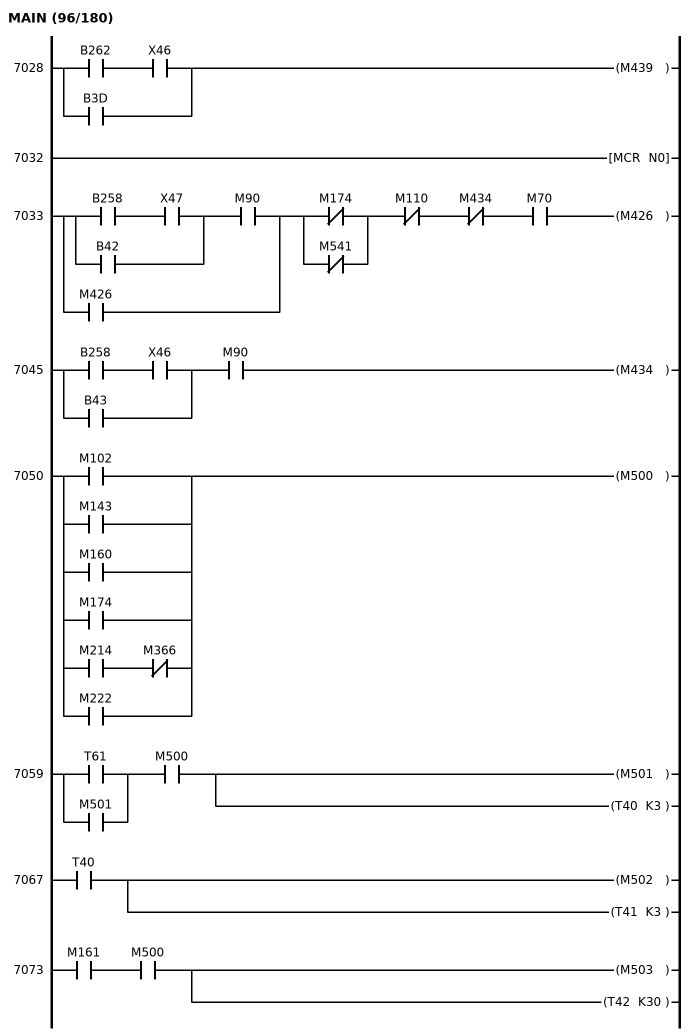
7028  LD      B262
      AND     X46
      OR      B3D
      OUT     M439
7032  MCR     N0
7033  LD      B258
      AND     X47
      OR      B42
      AND     M90
      OR      M426
      LDI     M174
      ORI     M541
      ANB
      ANI     M110
      ANI     M434
      AND     M70
      OUT     M426
7045  LD      B258
      AND     X46
      OR      B43
      AND     M90
      OUT     M434
7050  LD      M102
      OR      M143
      OR      M160
      OR      M174
      LD      M214
      ANI     M366
      ORB
      OR      M222
      OUT     M500
7059  LD      T61
      OR      M501
      AND     M500
      OUT     M501
      OUT     T40 K3
7067  LD      T40
      OUT     M502
      OUT     T41 K3
7073  LD      M161
      AND     M500
      OUT     M503
      OUT     T42 K30
